FUNCTION_BLOCK FB_Integer_To_BooleanArray
VAR_INPUT
	IntegerValue: INT := -1; // Inte value from Radiobutoon or whatever indexed component
	ArrayLength: INT := 2; // rquired length of the output Array 
END_VAR
VAR_OUTPUT
	OutputValue: ARRAY [0..1] OF BOOL; 
END_VAR
VAR
	i: INT;  // Loop counter
END_VAR

END_FUNCTION_BLOCK

(* stored: Version 1.1.0.1, ProductVersion 3.1.4024.12
   POU FB_Integer_To_BooleanArray: Id {9a7ffdf6-7ab1-4186-9a02-e79d8507b734}, SpecialFunc None *)
